SREFP 3 C00091 BC00091  +REFP EC00091
CALL JOB:SEARCH-R1-S13D
SET P023 P006
SFTON3D P023
SMOVL C00092 BC00092 V=166.7  +MOVJ EC00092
SMOVL C00093 BC00093 V=500.0  +MOVJ EC00093
SMOVL C00094 BC00094 V=166.7  +MOVJ EC00094
SREFP 3 C00095 BC00095  +REFP EC00095
CALL JOB:SEARCH-R1-S13D
SET P023 P006
SFTON3D P023
SMOVL C00096 BC00096 V=166.7  +MOVJ EC00096
SMOVL C00097 BC00097 V=166.7  +MOVJ EC00097
SREFP 3 C00098 BC00098  +REFP EC00098
CALL JOB:SEARCH-R1-S13D
SET P023 P006
SFTON3D P023
SMOVL C00099 BC00099 V=166.7  +MOVJ EC00099
MOVL C00100 BC00100 V=1000.0  +MOVJ EC00100 VJ=100.00
MOVJ C00101 BC00101 VJ=80.00  +MOVJ EC00101 VJ=80.00
MOVJ C00102 BC00102 VJ=80.00  +MOVJ EC00102 VJ=80.00
SFTOF3D
MOVJ C00103 BC00103 VJ=80.00  +MOVJ EC00103 VJ=80.00
SMOVL C00104 BC00104 V=166.7  +MOVJ EC00104
SREFP 3 C00105 BC00105  +REFP EC00105
CALL JOB:SEARCH-R1-S13D
SET P061 P006
SFTON3D P061
SMOVL C00106 BC00106 V=166.7  +MOVJ EC00106
SREFP 3 C00107 BC00107  +REFP EC00107
CALL JOB:SEARCH-R1-S13D
SET P061 P006
SFTON3D P061
SMOVL C00108 BC00108 V=166.7  +MOVJ EC00108
SFTOF3D
SMOVL C00109 BC00109 V=500.0  +MOVJ EC00109
SMOVL C00110 BC00110 V=166.7  +MOVJ EC00110
SREFP 3 C00111 BC00111  +REFP EC00111
CALL JOB:SEARCH-R1-S13D
SET P062 P006
SFTON3D P062
SMOVL C00112 BC00112 V=166.7  +MOVJ EC00112
SREFP 3 C00113 BC00113  +REFP EC00113
CALL JOB:SEARCH-R1-S13D
SET P062 P006
SFTON3D P062
SMOVL C00114 BC00114 V=166.7  +MOVJ EC00114
SFTOF3D
SMOVL C00115 BC00115 V=500.0  +MOVJ EC00115
SMOVL C00116 BC00116 V=166.7  +MOVJ EC00116
SREFP 3 C00117 BC00117  +REFP EC00117
CALL JOB:SEARCH-R1-S13D
SET P063 P006
SFTON3D P063
SMOVL C00118 BC00118 V=166.7  +MOVJ EC00118
SREFP 3 C00119 BC00119  +REFP EC00119
CALL JOB:SEARCH-R1-S13D
SET P063 P006
SFTON3D P063
SMOVL C00120 BC00120 V=166.7  +MOVJ EC00120
SFTOF3D
SMOVL C00121 BC00121 V=500.0  +MOVJ EC00121
MOVJ C00122 BC00122 VJ=80.00  +MOVJ EC00122 VJ=80.00
MOVJ C00123 BC00123 VJ=80.00  +MOVJ EC00123 VJ=80.00
'EndPath S3464
MOVJ C00124 BC00124 VJ=100.00  +MOVJ EC00124 VJ=100.00
'Path S3465
SFTOF3D
MOVJ C00125 BC00125 VJ=100.00  +MOVJ EC00125 VJ=100.00
MOVL C00126 BC00126 V=666.7  +MOVJ EC00126 VJ=100.00
SMOVL C00127 BC00127 V=166.7  +MOVJ EC00127
SREFP 3 C00128 BC00128  +REFP EC00128
CALL JOB:SEARCH-R1-S13D
SET P024 P006
SFTON3D P024
SMOVL C00129 BC00129 V=166.7  +MOVJ EC00129
SREFP 3 C00130 BC00130  +REFP EC00130
CALL JOB:SEARCH-R1-S13D
SET P024 P006
SFTON3D P024
SMOVL C00131 BC00131 V=166.7  +MOVJ EC00131
SMOVL C00132 BC00132 V=166.7  +MOVJ EC00132
SREFP 3 C00133 BC00133  +REFP EC00133
CALL JOB:SEARCH-R1-S13D
SET P024 P006
SFTON3D P024
SMOVL C00134 BC00134 V=166.7  +MOVJ EC00134
MOVL C00135 BC00135 V=1000.0  +MOVJ EC00135 VJ=100.00
'EndPath S3465
'Path S3476
SFTOF3D
MOVJ C00136 BC00136 VJ=100.00  +MOVJ EC00136 VJ=100.00
MOVL C00137 BC00137 V=666.7  +MOVJ EC00137 VJ=100.00
SMOVL C00138 BC00138 V=166.7  +MOVJ EC00138
SREFP 3 C00139 BC00139  +REFP EC00139
CALL JOB:SEARCH-R1-S13D
SET P035 P006
SFTON3D P035
SMOVL C00140 BC00140 V=166.7  +MOVJ EC00140
SREFP 3 C00141 BC00141  +REFP EC00141
CALL JOB:SEARCH-R1-S13D
SET P035 P006
SFTON3D P035
SMOVL C00142 BC00142 V=166.7  +MOVJ EC00142
SMOVL C00143 BC00143 V=333.3  +MOVJ EC00143
SMOVL C00144 BC00144 V=166.7  +MOVJ EC00144
SREFP 3 C00145 BC00145  +REFP EC00145
CALL JOB:SEARCH-R1-S13D
SET P035 P006
SFTON3D P035
SMOVL C00146 BC00146 V=166.7  +MOVJ EC00146
MOVL C00147 BC00147 V=1000.0  +MOVJ EC00147 VJ=100.00
'EndPath S3476
'Path S3470
SFTOF3D
MOVJ C00148 BC00148 VJ=100.00  +MOVJ EC00148 VJ=100.00
MOVL C00149 BC00149 V=666.7  +MOVJ EC00149 VJ=100.00
SMOVL C00150 BC00150 V=166.7  +MOVJ EC00150
SREFP 3 C00151 BC00151  +REFP EC00151
CALL JOB:SEARCH-R1-S13D
SET P029 P006
SFTON3D P029
SMOVL C00152 BC00152 V=166.7  +MOVJ EC00152
SREFP 3 C00153 BC00153  +REFP EC00153
CALL JOB:SEARCH-R1-S13D
SET P029 P006
SFTON3D P029
SMOVL C00154 BC00154 V=166.7  +MOVJ EC00154
SMOVL C00155 BC00155 V=250.0  +MOVJ EC00155
SMOVL C00156 BC00156 V=166.7  +MOVJ EC00156
SREFP 3 C00157 BC00157  +REFP EC00157
CALL JOB:SEARCH-R1-S13D
SET P029 P006
SFTON3D P029
SMOVL C00158 BC00158 V=166.7  +MOVJ EC00158
MOVL C00159 BC00159 V=1000.0  +MOVJ EC00159 VJ=100.00
'EndPath S3470
'Path S4850
SFTOF3D
MOVL C00160 BC00160 V=666.7  +MOVJ EC00160 VJ=100.00
SMOVL C00161 BC00161 V=166.7  +MOVJ EC00161
SREFP 3 C00162 BC00162  +REFP EC00162
CALL JOB:SEARCH-R1-S13D
SET P071 P006
SFTON3D P071
SMOVL C00163 BC00163 V=166.7  +MOVJ EC00163
SREFP 3 C00164 BC00164  +REFP EC00164
CALL JOB:SEARCH-R1-S13D
SET P071 P006
SFTON3D P071
SMOVL C00165 BC00165 V=166.7  +MOVJ EC00165
SMOVL C00166 BC00166 V=166.7  +MOVJ EC00166
SREFP 3 C00167 BC00167  +REFP EC00167
CALL JOB:SEARCH-R1-S13D
SET P071 P006
SFTON3D P071
SMOVL C00168 BC00168 V=166.7  +MOVJ EC00168
MOVL C00169 BC00169 V=1000.0  +MOVJ EC00169 VJ=100.00
'EndPath S4850
'Path S4851
SFTOF3D
MOVJ C00170 BC00170 VJ=100.00  +MOVJ EC00170 VJ=100.00
MOVL C00171 BC00171 V=666.7  +MOVJ EC00171 VJ=100.00
SMOVL C00172 BC00172 V=166.7  +MOVJ EC00172
SREFP 3 C00173 BC00173  +REFP EC00173
CALL JOB:SEARCH-R1-S13D
SET P072 P006
SFTON3D P072
SMOVL C00174 BC00174 V=166.7  +MOVJ EC00174
SREFP 3 C00175 BC00175  +REFP EC00175
CALL JOB:SEARCH-R1-S13D
SET P072 P006
SFTON3D P072
SMOVL C00176 BC00176 V=166.7  +MOVJ EC00176
MOVL C00177 BC00177 V=1000.0  +MOVJ EC00177 VJ=100.00
'EndPath S4851
MOVJ C00178 BC00178 VJ=100.00  +MOVJ EC00178 VJ=100.00
MOVJ C00179 BC00179 VJ=100.00  +MOVJ EC00179 VJ=100.00
'Path S4852
SFTOF3D
MOVJ C00180 BC00180 VJ=100.00  +MOVJ EC00180 VJ=100.00
MOVL C00181 BC00181 V=666.7  +MOVJ EC00181 VJ=100.00
SMOVL C00182 BC00182 V=166.7  +MOVJ EC00182
SREFP 3 C00183 BC00183  +REFP EC00183
CALL JOB:SEARCH-R1-S13D
SET P073 P006
SFTON3D P073
SMOVL C00184 BC00184 V=166.7  +MOVJ EC00184
SMOVL C00185 BC00185 V=166.7  +MOVJ EC00185
SREFP 3 C00186 BC00186  +REFP EC00186
CALL JOB:SEARCH-R1-S13D
SET P073 P006
SFTON3D P073
SMOVL C00187 BC00187 V=166.7  +MOVJ EC00187
SMOVL C00188 BC00188 V=166.7  +MOVJ EC00188
SREFP 3 C00189 BC00189  +REFP EC00189
CALL JOB:SEARCH-R1-S13D
SET P073 P006
SFTON3D P073
SMOVL C00190 BC00190 V=166.7  +MOVJ EC00190
MOVL C00191 BC00191 V=1000.0  +MOVJ EC00191 VJ=100.00
'EndPath S4852
MOVJ C00192 BC00192 VJ=100.00  +MOVJ EC00192 VJ=100.00
'Path S4853
SFTOF3D
MOVJ C00193 BC00193 VJ=100.00  +MOVJ EC00193 VJ=100.00
MOVL C00194 BC00194 V=666.7  +MOVJ EC00194 VJ=100.00
SMOVL C00195 BC00195 V=166.7  +MOVJ EC00195
SREFP 3 C00196 BC00196  +REFP EC00196
CALL JOB:SEARCH-R1-S13D
SET P074 P006
SFTON3D P074
SMOVL C00197 BC00197 V=166.7  +MOVJ EC00197
SREFP 3 C00198 BC00198  +REFP EC00198
CALL JOB:SEARCH-R1-S13D
SET P074 P006
SFTON3D P074
SMOVL C00199 BC00199 V=166.7  +MOVJ EC00199
MOVL C00200 BC00200 V=1000.0  +MOVJ EC00200 VJ=100.00
'EndPath S4853
'Path S3467
SFTOF3D
MOVJ C00201 BC00201 VJ=100.00  +MOVJ EC00201 VJ=100.00
MOVJ C00202 BC00202 VJ=50.00  +MOVJ EC00202 VJ=50.00
MOVJ C00203 BC00203 VJ=100.00  +MOVJ EC00203 VJ=100.00
MOVJ C00204 BC00204 VJ=100.00  +MOVJ EC00204 VJ=100.00
MOVL C00205 BC00205 V=666.7  +MOVJ EC00205 VJ=100.00
SMOVL C00206 BC00206 V=166.7  +MOVJ EC00206
SREFP 3 C00207 BC00207  +REFP EC00207
CALL JOB:SEARCH-R1-S13D
SET P026 P006
SFTON3D P026
SMOVL C00208 BC00208 V=166.7  +MOVJ EC00208
SREFP 3 C00209 BC00209  +REFP EC00209
CALL JOB:SEARCH-R1-S13D
SET P026 P006
SFTON3D P026
SMOVL C00210 BC00210 V=166.7  +MOVJ EC00210
SMOVL C00211 BC00211 V=800.0  +MOVJ EC00211
SMOVL C00212 BC00212 V=166.7  +MOVJ EC00212
SREFP 3 C00213 BC00213  +REFP EC00213
CALL JOB:SEARCH-R1-S13D
SET P026 P006
SFTON3D P026
SMOVL C00214 BC00214 V=166.7  +MOVJ EC00214
MOVL C00215 BC00215 V=1000.0  +MOVJ EC00215 VJ=100.00
'EndPath S3467
MOVJ C00216 BC00216 VJ=100.00  +MOVJ EC00216 VJ=100.00
'Path S3466
SFTOF3D
MOVJ C00217 BC00217 VJ=100.00  +MOVJ EC00217 VJ=100.00
MOVL C00218 BC00218 V=666.7  +MOVJ EC00218 VJ=100.00
SMOVL C00219 BC00219 V=166.7  +MOVJ EC00219
SREFP 3 C00220 BC00220  +REFP EC00220
CALL JOB:SEARCH-R1-S13D
SET P025 P006
SFTON3D P025
SMOVL C00221 BC00221 V=166.7  +MOVJ EC00221
SMOVL C00222 BC00222 V=166.7  +MOVJ EC00222
SREFP 3 C00223 BC00223  +REFP EC00223
CALL JOB:SEARCH-R1-S13D
SET P025 P006
SFTON3D P025
SMOVL C00224 BC00224 V=166.7  +MOVJ EC00224
SMOVL C00225 BC00225 V=200.0  +MOVJ EC00225
SMOVL C00226 BC00226 V=166.7  +MOVJ EC00226
SREFP 3 C00227 BC00227  +REFP EC00227
CALL JOB:SEARCH-R1-S13D
SET P025 P006
SFTON3D P025
SMOVL C00228 BC00228 V=166.7  +MOVJ EC00228
MOVL C00229 BC00229 V=1000.0  +MOVJ EC00229 VJ=100.00
'EndPath S3466
MOVJ C00230 BC00230 VJ=100.00  +MOVJ EC00230 VJ=100.00
'Path S3469
SFTOF3D
MOVJ C00231 BC00231 VJ=100.00  +MOVJ EC00231 VJ=100.00
MOVL C00232 BC00232 V=666.7  +MOVJ EC00232 VJ=100.00
SMOVL C00233 BC00233 V=166.7  +MOVJ EC00233
SREFP 3 C00234 BC00234  +REFP EC00234
CALL JOB:SEARCH-R1-S13D
SET P028 P006
SFTON3D P028
SMOVL C00235 BC00235 V=166.7  +MOVJ EC00235
SREFP 3 C00236 BC00236  +REFP EC00236
CALL JOB:SEARCH-R1-S13D
SET P028 P006
SFTON3D P028
SMOVL C00237 BC00237 V=166.7  +MOVJ EC00237
SMOVL C00238 BC00238 V=333.3  +MOVJ EC00238
SMOVL C00239 BC00239 V=166.7  +MOVJ EC00239
SREFP 3 C00240 BC00240  +REFP EC00240
CALL JOB:SEARCH-R1-S13D
SET P028 P006
SFTON3D P028
SMOVL C00241 BC00241 V=166.7  +MOVJ EC00241
MOVL C00242 BC00242 V=1000.0  +MOVJ EC00242 VJ=100.00
'EndPath S3469
MOVJ C00243 BC00243 VJ=100.00  +MOVJ EC00243 VJ=100.00
'Path S3474
SFTOF3D
MOVJ C00244 BC00244 VJ=100.00  +MOVJ EC00244 VJ=100.00
MOVL C00245 BC00245 V=666.7  +MOVJ EC00245 VJ=100.00
SMOVL C00246 BC00246 V=166.7  +MOVJ EC00246
SREFP 3 C00247 BC00247  +REFP EC00247
CALL JOB:SEARCH-R1-S13D
SET P033 P006
SFTON3D P033
SMOVL C00248 BC00248 V=166.7  +MOVJ EC00248
SREFP 3 C00249 BC00249  +REFP EC00249
CALL JOB:SEARCH-R1-S13D
SET P033 P006
SFTON3D P033
SMOVL C00250 BC00250 V=166.7  +MOVJ EC00250
SMOVL C00251 BC00251 V=250.0  +MOVJ EC00251
SMOVL C00252 BC00252 V=166.7  +MOVJ EC00252
SREFP 3 C00253 BC00253  +REFP EC00253
CALL JOB:SEARCH-R1-S13D
SET P033 P006
SFTON3D P033
SMOVL C00254 BC00254 V=166.7  +MOVJ EC00254
MOVL C00255 BC00255 V=1000.0  +MOVJ EC00255 VJ=100.00
'EndPath S3474
'Path S3468
SFTOF3D
MOVJ C00256 BC00256 VJ=100.00  +MOVJ EC00256 VJ=100.00
MOVL C00257 BC00257 V=666.7  +MOVJ EC00257 VJ=100.00
SMOVL C00258 BC00258 V=166.7  +MOVJ EC00258
SREFP 3 C00259 BC00259  +REFP EC00259
CALL JOB:SEARCH-R1-S13D
SET P027 P006
SFTON3D P027
SMOVL C00260 BC00260 V=166.7  +MOVJ EC00260
SMOVL C00261 BC00261 V=166.7  +MOVJ EC00261
SREFP 3 C00262 BC00262  +REFP EC00262
CALL JOB:SEARCH-R1-S13D
SET P027 P006
SFTON3D P027
SMOVL C00263 BC00263 V=166.7  +MOVJ EC00263
SMOVL C00264 BC00264 V=166.7  +MOVJ EC00264
SREFP 3 C00265 BC00265  +REFP EC00265
CALL JOB:SEARCH-R1-S13D
SET P027 P006
SFTON3D P027
SMOVL C00266 BC00266 V=166.7  +MOVJ EC00266
MOVL C00267 BC00267 V=1000.0  +MOVJ EC00267 VJ=100.00
'EndPath S3468
'Path S3471
SFTOF3D
MOVJ C00268 BC00268 VJ=100.00  +MOVJ EC00268 VJ=100.00
MOVL C00269 BC00269 V=666.7  +MOVJ EC00269 VJ=100.00
SMOVL C00270 BC00270 V=166.7  +MOVJ EC00270
SREFP 3 C00271 BC00271  +REFP EC00271
CALL JOB:SEARCH-R1-S13D
SET P030 P006
SFTON3D P030
SMOVL C00272 BC00272 V=166.7  +MOVJ EC00272
SREFP 3 C00273 BC00273  +REFP EC00273
CALL JOB:SEARCH-R1-S13D
SET P030 P006
SFTON3D P030
SMOVL C00274 BC00274 V=166.7  +MOVJ EC00274
MOVL C00275 BC00275 V=1000.0  +MOVJ EC00275 VJ=100.00
'EndPath S3471
'Path S3472
SFTOF3D
MOVJ C00276 BC00276 VJ=100.00  +MOVJ EC00276 VJ=100.00
MOVL C00277 BC00277 V=666.7  +MOVJ EC00277 VJ=100.00
SMOVL C00278 BC00278 V=166.7  +MOVJ EC00278
SREFP 3 C00279 BC00279  +REFP EC00279
CALL JOB:SEARCH-R1-S13D
SET P031 P006
SFTON3D P031
SMOVL C00280 BC00280 V=166.7  +MOVJ EC00280
SREFP 3 C00281 BC00281  +REFP EC00281
CALL JOB:SEARCH-R1-S13D
SET P031 P006
SFTON3D P031
SMOVL C00282 BC00282 V=166.7  +MOVJ EC00282
MOVL C00283 BC00283 V=1000.0  +MOVJ EC00283 VJ=100.00
'EndPath S3472
MOVJ C00284 BC00284 VJ=100.00  +MOVJ EC00284 VJ=100.00
'Path S3472
SFTOF3D
MOVJ C00285 BC00285 VJ=100.00  +MOVJ EC00285 VJ=100.00
MOVL C00286 BC00286 V=666.7  +MOVJ EC00286 VJ=100.00
SMOVL C00287 BC00287 V=166.7  +MOVJ EC00287
SREFP 3 C00288 BC00288  +REFP EC00288
CALL JOB:SEARCH-R1-S13D
SET P032 P006
SFTON3D P032
SMOVL C00289 BC00289 V=166.7  +MOVJ EC00289
SREFP 3 C00290 BC00290  +REFP EC00290
CALL JOB:SEARCH-R1-S13D
SET P032 P006
SFTON3D P032
SMOVL C00291 BC00291 V=166.7  +MOVJ EC00291
SMOVL C00292 BC00292 V=133.3  +MOVJ EC00292
SREFP 3 C00293 BC00293  +REFP EC00293
CALL JOB:SEARCH-R1-S13D
SET P032 P006
SFTON3D P032
SMOVL C00294 BC00294 V=166.7  +MOVJ EC00294
MOVL C00295 BC00295 V=1000.0  +MOVJ EC00295 VJ=100.00
'EndPath S3472
MOVJ C00296 BC00296 VJ=100.00  +MOVJ EC00296 VJ=100.00
'Path S3477
SFTOF3D
MOVJ C00297 BC00297 VJ=100.00  +MOVJ EC00297 VJ=100.00
SMOVL C00298 BC00298 V=166.7  +MOVJ EC00298
SREFP 3 C00299 BC00299  +REFP EC00299
CALL JOB:SEARCH-R1-S13D
SET P069 P006
SFTON3D P069
SMOVL C00300 BC00300 V=250.0  +MOVJ EC00300
SMOVL C00301 BC00301 V=250.0  +MOVJ EC00301
SMOVL C00302 BC00302 V=166.7  +MOVJ EC00302
SREFP 3 C00303 BC00303  +REFP EC00303
CALL JOB:SEARCH-R1-S13D
SET P069 P006
SFTON3D P069
SMOVL C00304 BC00304 V=166.7  +MOVJ EC00304
SFTOF3D
SMOVL C00305 BC00305 V=666.7  +MOVJ EC00305
MOVL C00306 BC00306 V=666.7  +MOVJ EC00306 VJ=100.00
SMOVL C00307 BC00307 V=166.7  +MOVJ EC00307
SREFP 3 C00308 BC00308  +REFP EC00308
CALL JOB:SEARCH-R1-S13D
SET P052 P006
SFTON3D P052
SMOVL C00309 BC00309 V=166.7  +MOVJ EC00309
SREFP 3 C00310 BC00310  +REFP EC00310
CALL JOB:SEARCH-R1-S13D
SET P052 P006
SFTON3D P052
SMOVL C00311 BC00311 V=166.7  +MOVJ EC00311
MOVL C00312 BC00312 V=1000.0  +MOVJ EC00312 VJ=100.00
'EndPath S3477
MOVJ C00313 BC00313 VJ=100.00  +MOVJ EC00313 VJ=100.00
'poprawiÄ searcha- nie mialem
'wyciecia
'Path S3478
SFTOF3D
MOVJ C00314 BC00314 VJ=100.00  +MOVJ EC00314 VJ=100.00
MOVL C00315 BC00315 V=666.7  +MOVJ EC00315 VJ=100.00
SMOVL C00316 BC00316 V=166.7  +MOVJ EC00316
SREFP 3 C00317 BC00317  +REFP EC00317
CALL JOB:SEARCH-R1-S13D
SET P053 P006
SFTON3D P053
SMOVL C00318 BC00318 V=166.7  +MOVJ EC00318
SREFP 3 C00319 BC00319  +REFP EC00319
CALL JOB:SEARCH-R1-S13D
SET P053 P006
SFTON3D P053
SMOVL C00320 BC00320 V=166.7  +MOVJ EC00320
MOVL C00321 BC00321 V=1000.0  +MOVJ EC00321 VJ=100.00
'EndPath S3478
'
MOVJ C00322 BC00322 VJ=100.00  +MOVJ EC00322 VJ=100.00
'Path W3476
SFTOF3D
SFTON3D P033
MOVJ C00323 BC00323 VJ=100.00  +MOVJ EC00323 VJ=100.00
SMOVL C00324 BC00324 V=800.0  +MOVJ EC00324
SMOVL C00325 BC00325 V=166.7 PL=0  +MOVJ EC00325
MACRO1 MJ#(0) ARGF14
ARCON
SMOVL C00326 BC00326 V=10.0  +MOVJ EC00326
ARCOF
SMOVL C00327 BC00327 V=800.0  +MOVJ EC00327
SMOVL C00328 BC00328 V=1000.0  +MOVJ EC00328
SFTOF3D
'EndPath W3476
'Path W3477
SFTOF3D
SFTON3D P033
MOVJ C00329 BC00329 VJ=100.00  +MOVJ EC00329 VJ=100.00
SMOVL C00330 BC00330 V=800.0  +MOVJ EC00330
SMOVL C00331 BC00331 V=166.7 PL=0  +MOVJ EC00331
SMOVL C00332 BC00332 V=10.0  +MOVJ EC00332
SMOVL C00333 BC00333 V=10.0  +MOVJ EC00333
SMOVL C00334 BC00334 V=10.0  +MOVJ EC00334
ARCOF
SMOVL C00335 BC00335 V=800.0  +MOVJ EC00335
SMOVL C00336 BC00336 V=1000.0  +MOVJ EC00336
SFTOF3D
'EndPath W3477
MOVJ C00337 BC00337 VJ=100.00  +MOVJ EC00337 VJ=100.00
'Path W3478
SFTOF3D
SFTON3D P033
MOVJ C00338 BC00338 VJ=100.00  +MOVJ EC00338 VJ=100.00
SMOVL C00339 BC00339 V=800.0  +MOVJ EC00339
SMOVL C00340 BC00340 V=166.7 PL=0  +MOVJ EC00340
ARCON
SMOVL C00341 BC00341 V=10.0  +MOVJ EC00341
SMOVL C00342 BC00342 V=10.0  +MOVJ EC00342
SMOVL C00343 BC00343 V=10.0  +MOVJ EC00343
ARCOF
SMOVL C00344 BC00344 V=800.0  +MOVJ EC00344
SMOVL C00345 BC00345 V=1000.0  +MOVJ EC00345
SFTOF3D
'EndPath W3478
MOVJ C00346 BC00346 VJ=100.00  +MOVJ EC00346 VJ=100.00
MOVJ C00347 BC00347 VJ=100.00  +MOVJ EC00347 VJ=100.00
'9
'Path W3479
SFTOF3D
SFTON3D P026
MOVJ C00348 BC00348 VJ=100.00  +MOVJ EC00348 VJ=100.00
SMOVL C00349 BC00349 V=800.0  +MOVJ EC00349
SMOVL C00350 BC00350 V=166.7 PL=0  +MOVJ EC00350
ARCON
SMOVL C00351 BC00351 V=9.2  +MOVJ EC00351
SMOVL C00352 BC00352 V=9.2  +MOVJ EC00352
SMOVL C00353 BC00353 V=9.2  +MOVJ EC00353
ARCOF
SMOVL C00354 BC00354 V=800.0  +MOVJ EC00354
SMOVL C00355 BC00355 V=1000.0  +MOVJ EC00355
SFTOF3D
'EndPath W3479
'Path W3480
SFTOF3D
SFTON3D P026
MOVJ C00356 BC00356 VJ=100.00  +MOVJ EC00356 VJ=100.00
SMOVL C00357 BC00357 V=800.0  +MOVJ EC00357
SMOVL C00358 BC00358 V=150.0 PL=0  +MOVJ EC00358
ARCON
SMOVL C00359 BC00359 V=10.0  +MOVJ EC00359
SMOVL C00360 BC00360 V=10.0  +MOVJ EC00360
SMOVL C00361 BC00361 V=10.0  +MOVJ EC00361
ARCOF
SMOVL C00362 BC00362 V=800.0  +MOVJ EC00362
SMOVL C00363 BC00363 V=1000.0  +MOVJ EC00363
SFTOF3D
'EndPath W3480
'Path W3481
SFTOF3D
SFTON3D P026
MOVJ C00364 BC00364 VJ=100.00  +MOVJ EC00364 VJ=100.00
SMOVL C00365 BC00365 V=800.0  +MOVJ EC00365
SMOVL C00366 BC00366 V=150.0 PL=0  +MOVJ EC00366
SMOVL C00367 BC00367 V=10.0  +MOVJ EC00367
ARCOF
SMOVL C00368 BC00368 V=800.0  +MOVJ EC00368
SMOVL C00369 BC00369 V=1000.0  +MOVJ EC00369
SFTOF3D
'EndPath W3481
MOVJ C00370 BC00370 VJ=100.00  +MOVJ EC00370 VJ=100.00
'uwaga na podajnik
'Path W3481
SFTOF3D
SFTON3D P026
MOVJ C00371 BC00371 VJ=50.00  +MOVJ EC00371 VJ=15.00
SMOVL C00372 BC00372 V=800.0  +MOVJ EC00372
SMOVL C00373 BC00373 V=150.0 PL=0  +MOVJ EC00373
ARCON
SMOVL C00374 BC00374 V=10.0  +MOVJ EC00374
SMOVL C00375 BC00375 V=10.0  +MOVJ EC00375
ARCOF
SMOVL C00376 BC00376 V=800.0  +MOVJ EC00376
SMOVL C00377 BC00377 V=1000.0  +MOVJ EC00377
SFTOF3D
'EndPath W3481
'brak dostepu offset drutu 1cm
'Path W3482
SFTOF3D
SFTON3D P026
MOVJ C00378 BC00378 VJ=100.00  +MOVJ EC00378 VJ=100.00
SMOVL C00379 BC00379 V=800.0  +MOVJ EC00379
SMOVL C00380 BC00380 V=150.0 PL=0  +MOVJ EC00380
ARCON
SMOVL C00381 BC00381 V=10.0  +MOVJ EC00381
ARCOF
SMOVL C00382 BC00382 V=800.0  +MOVJ EC00382
SMOVL C00383 BC00383 V=1000.0  +MOVJ EC00383
SFTOF3D
'EndPath W3482
MOVJ C00384 BC00384 VJ=100.00  +MOVJ EC00384 VJ=100.00
MOVJ C00385 BC00385 VJ=100.00  +MOVJ EC00385 VJ=100.00
'10
'11
'Path W3484
SFTOF3D
SFTON3D P025
MOVJ C00386 BC00386 VJ=100.00  +MOVJ EC00386 VJ=100.00
SMOVL C00387 BC00387 V=800.0  +MOVJ EC00387
SMOVL C00388 BC00388 V=150.0 PL=0  +MOVJ EC00388
ARCON
SMOVL C00389 BC00389 V=10.0  +MOVJ EC00389
SMOVL C00390 BC00390 V=10.0  +MOVJ EC00390
ARCOF
SMOVL C00391 BC00391 V=800.0  +MOVJ EC00391
SMOVL C00392 BC00392 V=1000.0  +MOVJ EC00392
SFTOF3D
'EndPath W3484
MOVJ C00393 BC00393 VJ=100.00  +MOVJ EC00393 VJ=100.00
'brak dostepu offset drutu 1cm
'Path W3483
SFTOF3D
SFTON3D P025
MOVJ C00394 BC00394 VJ=100.00  +MOVJ EC00394 VJ=100.00
SMOVL C00395 BC00395 V=800.0  +MOVJ EC00395
SMOVL C00396 BC00396 V=166.7 PL=0  +MOVJ EC00396
ARCON
SMOVL C00397 BC00397 V=10.0  +MOVJ EC00397
ARCOF
SMOVL C00398 BC00398 V=800.0  +MOVJ EC00398
SMOVL C00399 BC00399 V=1000.0  +MOVJ EC00399
SFTOF3D
'EndPath W3483
MOVJ C00400 BC00400 VJ=100.00  +MOVJ EC00400 VJ=100.00
MOVJ C00401 BC00401 VJ=100.00  +MOVJ EC00401 VJ=100.00
MOVJ C00402 BC00402 VJ=100.00  +MOVJ EC00402 VJ=100.00
'Path W4854
SFTOF3D
SFTON3D P073
MOVJ C00403 BC00403 VJ=100.00  +MOVJ EC00403 VJ=100.00
SMOVL C00404 BC00404 V=800.0  +MOVJ EC00404
SMOVL C00405 BC00405 V=150.0 PL=0  +MOVJ EC00405
MACRO1 MJ#(0) ARGF9
ARCON
SMOVL C00406 BC00406 V=9.2  +MOVJ EC00406
SFTON3D P074
SMOVL C00407 BC00407 V=9.2  +MOVJ EC00407
SMOVL C00408 BC00408 V=9.2  +MOVJ EC00408
ARCOF
SMOVL C00409 BC00409 V=800.0  +MOVJ EC00409
SMOVL C00410 BC00410 V=1000.0  +MOVJ EC00410
SFTOF3D
'EndPath W4854
'12
MOVJ C00411 BC00411 VJ=100.00  +MOVJ EC00411 VJ=100.00
MOVJ C00412 BC00412 VJ=100.00  +MOVJ EC00412 VJ=100.00
MOVJ C00413 BC00413 VJ=100.00  +MOVJ EC00413 VJ=100.00
'Path W3485
SFTOF3D
SFTON3D P034
MOVJ C00414 BC00414 VJ=100.00  +MOVJ EC00414 VJ=100.00
SMOVL C00415 BC00415 V=800.0  +MOVJ EC00415
SMOVL C00416 BC00416 V=150.0 PL=0  +MOVJ EC00416
MACRO1 MJ#(0) ARGF14
ARCON
SMOVL C00417 BC00417 V=10.0  +MOVJ EC00417
SMOVL C00418 BC00418 V=10.0  +MOVJ EC00418
SMOVL C00419 BC00419 V=10.0  +MOVJ EC00419
ARCOF
SMOVL C00420 BC00420 V=800.0  +MOVJ EC00420
SMOVL C00421 BC00421 V=1000.0  +MOVJ EC00421
SFTOF3D
MOVJ C00422 BC00422 VJ=80.00  +MOVJ EC00422 VJ=80.00
MOVJ C00423 BC00423 VJ=80.00  +MOVJ EC00423 VJ=80.00
MOVJ C00424 BC00424 VJ=80.00  +MOVJ EC00424 VJ=80.00
MACRO1 MJ#(0) ARGF6
SFTON3D P063
SMOVL C00425 BC00425 V=166.7  +MOVJ EC00425
ARCON
SMOVL C00426 BC00426 V=11.7  +MOVJ EC00426
SMOVL C00427 BC00427 V=11.7  +MOVJ EC00427
SFTON3D P062
SMOVL C00428 BC00428 V=11.0  +MOVJ EC00428
SMOVL C00429 BC00429 V=11.0  +MOVJ EC00429
SFTON3D P061
SMOVL C00430 BC00430 V=11.0  +MOVJ EC00430
SMOVL C00431 BC00431 V=11.0  +MOVJ EC00431
ARCOF
SMOVL C00432 BC00432 V=800.0  +MOVJ EC00432
SFTOF3D
MOVJ C00433 BC00433 VJ=80.00  +MOVJ EC00433 VJ=80.00
MOVJ C00434 BC00434 VJ=80.00  +MOVJ EC00434 VJ=80.00
MOVJ C00435 BC00435 VJ=80.00  +MOVJ EC00435 VJ=80.00
'EndPath W3485
'Path W3486
SFTOF3D
SFTON3D P050
MOVJ C00436 BC00436 VJ=100.00  +MOVJ EC00436 VJ=100.00
SMOVL C00437 BC00437 V=800.0  +MOVJ EC00437
SMOVL C00438 BC00438 V=150.0 PL=0  +MOVJ EC00438
MACRO1 MJ#(0) ARGF14
ARCON
SMOVL C00439 BC00439 V=10.0  +MOVJ EC00439
SMOVL C00440 BC00440 V=10.0  +MOVJ EC00440
SMOVL C00441 BC00441 V=10.0  +MOVJ EC00441
ARCOF
SMOVL C00442 BC00442 V=800.0  +MOVJ EC00442
SMOVL C00443 BC00443 V=1000.0  +MOVJ EC00443
SFTOF3D
'EndPath W3486
MOVJ C00444 BC00444 VJ=100.00  +MOVJ EC00444 VJ=100.00
'Path W3485
SFTOF3D
SFTON3D P034
MOVJ C00445 BC00445 VJ=100.00  +MOVJ EC00445 VJ=100.00
SMOVL C00446 BC00446 V=800.0  +MOVJ EC00446
SMOVL C00447 BC00447 V=166.7 PL=0  +MOVJ EC00447
ARCON
SMOVL C00448 BC00448 V=9.2  +MOVJ EC00448
SMOVL C00449 BC00449 V=9.2  +MOVJ EC00449
SMOVL C00450 BC00450 V=9.2  +MOVJ EC00450
ARCOF
SMOVL C00451 BC00451 V=800.0  +MOVJ EC00451
SMOVL C00452 BC00452 V=1000.0  +MOVJ EC00452
SFTOF3D
'EndPath W3485
'Path W3487
SFTOF3D
SFTON3D P054
MOVJ C00453 BC00453 VJ=100.00  +MOVJ EC00453 VJ=100.00
SMOVL C00454 BC00454 V=800.0  +MOVJ EC00454
SMOVL C00455 BC00455 V=150.0 PL=0  +MOVJ EC00455
ARCON
SMOVL C00456 BC00456 V=9.2  +MOVJ EC00456
SMOVL C00457 BC00457 V=9.2  +MOVJ EC00457
SMOVL C00458 BC00458 V=9.2  +MOVJ EC00458
ARCOF
SMOVL C00459 BC00459 V=800.0  +MOVJ EC00459
SMOVL C00460 BC00460 V=1000.0  +MOVJ EC00460
SFTOF3D
'EndPath W3487
MOVJ C00461 BC00461 VJ=100.00  +MOVJ EC00461 VJ=100.00
'Path W3487
SFTOF3D
SFTON3D P028
MOVJ C00462 BC00462 VJ=100.00  +MOVJ EC00462 VJ=100.00
SMOVL C00463 BC00463 V=800.0  +MOVJ EC00463
SMOVL C00464 BC00464 V=150.0 PL=0  +MOVJ EC00464
ARCON
SMOVL C00465 BC00465 V=9.2  +MOVJ EC00465
SMOVL C00466 BC00466 V=9.2  +MOVJ EC00466
SMOVL C00467 BC00467 V=9.2  +MOVJ EC00467
ARCOF
SMOVL C00468 BC00468 V=800.0  +MOVJ EC00468
SMOVL C00469 BC00469 V=1000.0  +MOVJ EC00469
SFTOF3D
'EndPath W3487
MOVJ C00470 BC00470 VJ=100.00  +MOVJ EC00470 VJ=100.00
MOVJ C00471 BC00471 VJ=100.00  +MOVJ EC00471 VJ=100.00
'brak dostepu offset 5mm
'Path W3488
SFTOF3D
SFTON3D P028
MOVJ C00472 BC00472 VJ=100.00  +MOVJ EC00472 VJ=100.00
SMOVL C00473 BC00473 V=800.0  +MOVJ EC00473
SMOVL C00474 BC00474 V=150.0 PL=0  +MOVJ EC00474
ARCON
SMOVL C00475 BC00475 V=11.7  +MOVJ EC00475
ARCOF
SMOVL C00476 BC00476 V=800.0  +MOVJ EC00476
SMOVL C00477 BC00477 V=1000.0  +MOVJ EC00477
SFTOF3D
'EndPath W3488
MOVJ C00478 BC00478 VJ=100.00  +MOVJ EC00478 VJ=100.00
'13
'Path W3489
SFTOF3D
SFTON3D P030
MOVJ C00479 BC00479 VJ=100.00  +MOVJ EC00479 VJ=100.00
SMOVL C00480 BC00480 V=800.0  +MOVJ EC00480
SMOVL C00481 BC00481 V=150.0 PL=0  +MOVJ EC00481
MACRO1 MJ#(0) ARGF9
ARCON
SWVON WEV#(10)
SFTON3D P031
SMOVL C00482 BC00482 V=12.5  +MOVJ EC00482
ARCOF
SWVOF
SMOVL C00483 BC00483 V=800.0  +MOVJ EC00483
SMOVL C00484 BC00484 V=1000.0  +MOVJ EC00484
SFTOF3D
'EndPath W3489
'Path W3490
SFTOF3D
MOVJ C00485 BC00485 VJ=100.00  +MOVJ EC00485 VJ=100.00
MACRO1 MJ#(0) ARGF6
SFTON3D P069
SMOVL C00486 BC00486 V=250.0  +MOVJ EC00486
ARCON
SMOVL C00487 BC00487 V=11.7  +MOVJ EC00487
ARCOF
SMOVL C00488 BC00488 V=250.0  +MOVJ EC00488
SFTOF3D
SFTON3D P052
MOVJ C00489 BC00489 VJ=100.00  +MOVJ EC00489 VJ=100.00
SMOVL C00490 BC00490 V=800.0  +MOVJ EC00490
SMOVL C00491 BC00491 V=150.0 PL=0  +MOVJ EC00491
MACRO1 MJ#(0) ARGF14
ARCON
SMOVL C00492 BC00492 V=10.0  +MOVJ EC00492
SMOVL C00493 BC00493 V=10.0  +MOVJ EC00493
SMOVL C00494 BC00494 V=10.0  +MOVJ EC00494
ARCOF
SMOVL C00495 BC00495 V=800.0  +MOVJ EC00495
SMOVL C00496 BC00496 V=1000.0  +MOVJ EC00496
SFTOF3D
'EndPath W3490
MOVJ C00497 BC00497 VJ=100.00  +MOVJ EC00497 VJ=100.00
'poprawic spoine - nie mialem w
'yciecia
'Path W3491
SFTOF3D
SFTON3D P053
MOVJ C00498 BC00498 VJ=100.00  +MOVJ EC00498 VJ=100.00
SMOVL C00499 BC00499 V=800.0  +MOVJ EC00499
SMOVL C00500 BC00500 V=150.0 PL=0  +MOVJ EC00500
ARCON
SMOVL C00501 BC00501 V=10.0  +MOVJ EC00501
SMOVL C00502 BC00502 V=10.0  +MOVJ EC00502
SMOVL C00503 BC00503 V=10.0  +MOVJ EC00503
ARCOF
SMOVL C00504 BC00504 V=800.0  +MOVJ EC00504
SMOVL C00505 BC00505 V=1000.0  +MOVJ EC00505
SFTOF3D
'EndPath W3491
'14
'15-brak
MOVJ C00506 BC00506 VJ=100.00  +MOVJ EC00506 VJ=100.00
'16
'Path W3491
SFTOF3D
SFTON3D P029
MOVJ C00507 BC00507 VJ=100.00  +MOVJ EC00507 VJ=100.00
SMOVL C00508 BC00508 V=800.0  +MOVJ EC00508
SMOVL C00509 BC00509 V=150.0 PL=0  +MOVJ EC00509
ARCON
SMOVL C00510 BC00510 V=10.0  +MOVJ EC00510
SMOVL C00511 BC00511 V=10.0  +MOVJ EC00511
ARCOF
SMOVL C00512 BC00512 V=800.0  +MOVJ EC00512
SMOVL C00513 BC00513 V=1000.0  +MOVJ EC00513
SFTOF3D
'EndPath W3491
MOVJ C00514 BC00514 VJ=100.00  +MOVJ EC00514 VJ=100.00
'Path W3492
SFTOF3D
SFTON3D P029
MOVJ C00515 BC00515 VJ=100.00  +MOVJ EC00515 VJ=100.00
SMOVL C00516 BC00516 V=800.0  +MOVJ EC00516
SMOVL C00517 BC00517 V=150.0 PL=0  +MOVJ EC00517
ARCON
SMOVL C00518 BC00518 V=10.0  +MOVJ EC00518
ARCOF
SMOVL C00519 BC00519 V=800.0  +MOVJ EC00519
SMOVL C00520 BC00520 V=1000.0  +MOVJ EC00520
SFTOF3D
'EndPath W3492
MOVJ C00521 BC00521 VJ=100.00  +MOVJ EC00521 VJ=100.00
MOVJ C00522 BC00522 VJ=100.00  +MOVJ EC00522 VJ=100.00
'Path W3493
SFTOF3D
SFTON3D P029
MOVJ C00523 BC00523 VJ=100.00  +MOVJ EC00523 VJ=100.00
SMOVL C00524 BC00524 V=800.0  +MOVJ EC00524
SMOVL C00525 BC00525 V=150.0 PL=0  +MOVJ EC00525
ARCON
SMOVL C00526 BC00526 V=10.0  +MOVJ EC00526
SMOVL C00527 BC00527 V=10.0  +MOVJ EC00527
SMOVL C00528 BC00528 V=10.0  +MOVJ EC00528
ARCON
SMOVL C00529 BC00529 V=11.7  +MOVJ EC00529
ARCON
SMOVL C00530 BC00530 V=11.7  +MOVJ EC00530
ARCOF
SMOVL C00531 BC00531 V=800.0  +MOVJ EC00531
SMOVL C00532 BC00532 V=1000.0  +MOVJ EC00532
SFTOF3D
'EndPath W3493
MOVJ C00533 BC00533 VJ=100.00  +MOVJ EC00533 VJ=100.00
MOVJ C00534 BC00534 VJ=100.00  +MOVJ EC00534 VJ=100.00
'17
'Path W3494
SFTOF3D
SFTON3D P027
MOVJ C00535 BC00535 VJ=100.00  +MOVJ EC00535 VJ=100.00
SMOVL C00536 BC00536 V=800.0  +MOVJ EC00536
SMOVL C00537 BC00537 V=150.0 PL=0  +MOVJ EC00537
ARCON
SMOVL C00538 BC00538 V=10.0  +MOVJ EC00538
ARCOF
SMOVL C00539 BC00539 V=800.0  +MOVJ EC00539
SMOVL C00540 BC00540 V=1000.0  +MOVJ EC00540
SFTOF3D
'EndPath W3494
'Path W3495
SFTOF3D
SFTON3D P027
MOVJ C00541 BC00541 VJ=100.00  +MOVJ EC00541 VJ=100.00
SMOVL C00542 BC00542 V=800.0  +MOVJ EC00542
SMOVL C00543 BC00543 V=150.0 PL=0  +MOVJ EC00543
ARCON
SMOVL C00544 BC00544 V=10.8  +MOVJ EC00544
ARCOF
SMOVL C00545 BC00545 V=800.0  +MOVJ EC00545
SMOVL C00546 BC00546 V=1000.0  +MOVJ EC00546
SFTOF3D
'EndPath W3495
'Path W3496
SFTOF3D
SFTON3D P027
MOVJ C00547 BC00547 VJ=100.00  +MOVJ EC00547 VJ=100.00
SFTOF3D
'EndPath W3496
MOVJ C00548 BC00548 VJ=100.00  +MOVJ EC00548 VJ=100.00
MOVJ C00549 BC00549 VJ=100.00  +MOVJ EC00549 VJ=100.00
MOVJ C00550 BC00550 VJ=100.00  +MOVJ EC00550 VJ=100.00
'18
'Path W3497
SFTOF3D
SFTON3D P024
MOVJ C00551 BC00551 VJ=100.00  +MOVJ EC00551 VJ=100.00
SMOVL C00552 BC00552 V=800.0  +MOVJ EC00552
SMOVL C00553 BC00553 V=150.0 PL=0  +MOVJ EC00553
ARCON
SMOVL C00554 BC00554 V=9.2  +MOVJ EC00554
SMOVL C00555 BC00555 V=9.2  +MOVJ EC00555
SMOVL C00556 BC00556 V=9.2  +MOVJ EC00556
SMOVL C00557 BC00557 V=9.2  +MOVJ EC00557
ARCOF
SMOVL C00558 BC00558 V=800.0  +MOVJ EC00558
SMOVL C00559 BC00559 V=1000.0  +MOVJ EC00559
SFTOF3D
'EndPath W3497
'
'Path W4855
SFTOF3D
SFTON3D P071
MOVJ C00560 BC00560 VJ=100.00  +MOVJ EC00560 VJ=100.00
SMOVL C00561 BC00561 V=800.0  +MOVJ EC00561
MACRO1 MJ#(0) ARGF9
SMOVL C00562 BC00562 V=150.0 PL=0  +MOVJ EC00562
ARCON
SMOVL C00563 BC00563 V=8.8  +MOVJ EC00563
SFTON3D P072
SMOVL C00564 BC00564 V=8.8  +MOVJ EC00564
SMOVL C00565 BC00565 V=8.8  +MOVJ EC00565
ARCOF
SMOVL C00566 BC00566 V=800.0  +MOVJ EC00566
SMOVL C00567 BC00567 V=1000.0  +MOVJ EC00567
SFTOF3D
'EndPath W4855
'
'
MOVJ C00568 BC00568 VJ=100.00  +MOVJ EC00568 VJ=100.00
'19
MOVJ C00569 BC00569 VJ=100.00  +MOVJ EC00569 VJ=100.00
'Path W3499
SFTOF3D
SFTON3D P023
MOVJ C00570 BC00570 VJ=100.00  +MOVJ EC00570 VJ=100.00
SMOVL C00571 BC00571 V=800.0  +MOVJ EC00571
SMOVL C00572 BC00572 V=150.0 PL=0  +MOVJ EC00572
MACRO1 MJ#(0) ARGF6
ARCON
SWVON WEV#(66)
SMOVL C00573 BC00573 V=7.5  +MOVJ EC00573
SMOVL C00574 BC00574 V=7.5  +MOVJ EC00574
SMOVL C00575 BC00575 V=7.5  +MOVJ EC00575
ARCOF
SWVOF
SMOVL C00576 BC00576 V=800.0  +MOVJ EC00576
SMOVL C00577 BC00577 V=1000.0  +MOVJ EC00577
SFTOF3D
'EndPath W3499
MOVJ C00578 BC00578 VJ=100.00  +MOVJ EC00578 VJ=100.00
'Path W3500
SFTOF3D
SFTON3D P034
MOVJ C00579 BC00579 VJ=100.00  +MOVJ EC00579 VJ=100.00
SMOVL C00580 BC00580 V=800.0  +MOVJ EC00580
MACRO1 MJ#(0) ARGF9
SMOVL C00581 BC00581 V=150.0 PL=0  +MOVJ EC00581
ARCON
SMOVL C00582 BC00582 V=8.3  +MOVJ EC00582
SFTON3D P050
SMOVL C00583 BC00583 V=8.3  +MOVJ EC00583
SMOVL C00584 BC00584 V=8.3  +MOVJ EC00584
ARCOF
SMOVL C00585 BC00585 V=800.0  +MOVJ EC00585
SMOVL C00586 BC00586 V=1000.0  +MOVJ EC00586
SFTOF3D
'EndPath W3500
'Path W3501
SFTOF3D
SFTON3D P051
MOVJ C00587 BC00587 VJ=100.00  +MOVJ EC00587 VJ=100.00
SMOVL C00588 BC00588 V=800.0  +MOVJ EC00588
SMOVL C00589 BC00589 V=150.0 PL=0  +MOVJ EC00589
ARCON
SWVON WEV#(60)
SMOVL C00590 BC00590 V=7.5  +MOVJ EC00590
SMOVL C00591 BC00591 V=7.5  +MOVJ EC00591
SMOVL C00592 BC00592 V=7.5  +MOVJ EC00592
ARCOF
SWVOF
SMOVL C00593 BC00593 V=800.0  +MOVJ EC00593
SMOVL C00594 BC00594 V=1000.0  +MOVJ EC00594
SFTOF3D
'EndPath W3501
MOVJ C00595 BC00595 VJ=100.00  +MOVJ EC00595 VJ=100.00
'20
MOVJ C00596 BC00596 VJ=100.00  +MOVJ EC00596 VJ=100.00
MOVJ C00597 BC00597 VJ=100.00  +MOVJ EC00597 VJ=100.00
'offset 5mm
'Path W3500
SFTOF3D
SFTON3D P032
MOVJ C00598 BC00598 VJ=100.00  +MOVJ EC00598 VJ=100.00
SMOVL C00599 BC00599 V=800.0  +MOVJ EC00599
SMOVL C00600 BC00600 V=150.0 PL=0  +MOVJ EC00600
ARCON
SMOVL C00601 BC00601 V=9.2  +MOVJ EC00601
ARCOF
SMOVL C00602 BC00602 V=800.0  +MOVJ EC00602
SMOVL C00603 BC00603 V=1000.0  +MOVJ EC00603
SFTOF3D
'EndPath W3500
SFTOF3D
'EndPath W3502
'offset 5mm
'Path W3503
SFTOF3D
SFTON3D P032
MOVJ C00604 BC00604 VJ=100.00  +MOVJ EC00604 VJ=100.00
SMOVL C00605 BC00605 V=800.0  +MOVJ EC00605
SMOVL C00606 BC00606 V=150.0 PL=0  +MOVJ EC00606
ARCON
SMOVL C00607 BC00607 V=10.0  +MOVJ EC00607
ARCOF
SMOVL C00608 BC00608 V=800.0  +MOVJ EC00608
SMOVL C00609 BC00609 V=1000.0  +MOVJ EC00609
SFTOF3D
'EndPath W3503
MOVJ C00610 BC00610 VJ=100.00  +MOVJ EC00610 VJ=100.00
'Path W3504
SFTOF3D
SFTON3D P032
MOVJ C00611 BC00611 VJ=100.00  +MOVJ EC00611 VJ=100.00
SMOVL C00612 BC00612 V=800.0  +MOVJ EC00612
SMOVL C00613 BC00613 V=150.0 PL=0  +MOVJ EC00613
ARCON
SMOVL C00614 BC00614 V=11.7  +MOVJ EC00614
SMOVL C00615 BC00615 V=11.7  +MOVJ EC00615
ARCOF
SMOVL C00616 BC00616 V=800.0  +MOVJ EC00616
SMOVL C00617 BC00617 V=1000.0  +MOVJ EC00617
SFTOF3D
'EndPath W3504
MOVJ C00618 BC00618 VJ=100.00  +MOVJ EC00618 VJ=100.00
'21
MOVJ C00619 BC00619 VJ=100.00  +MOVJ EC00619 VJ=100.00
'Path W3505
SFTOF3D
SFTON3D P021
MOVJ C00620 BC00620 VJ=100.00  +MOVJ EC00620 VJ=100.00
SMOVL C00621 BC00621 V=800.0  +MOVJ EC00621
SMOVL C00622 BC00622 V=150.0 PL=0  +MOVJ EC00622
ARCON
SFTON3D P022
SMOVL C00623 BC00623 V=10.8  +MOVJ EC00623
SMOVL C00624 BC00624 V=11.7  +MOVJ EC00624
ARCOF
SMOVL C00625 BC00625 V=800.0  +MOVJ EC00625
SMOVL C00626 BC00626 V=1000.0  +MOVJ EC00626
SFTOF3D
'EndPath W3505
MOVJ C00627 BC00627 VJ=100.00  +MOVJ EC00627 VJ=100.00
'Path W3506
SFTOF3D
SFTON3D P095
MOVJ C00628 BC00628 VJ=100.00  +MOVJ EC00628 VJ=100.00
SMOVL C00629 BC00629 V=800.0  +MOVJ EC00629
SMOVL C00630 BC00630 V=150.0 PL=0  +MOVJ EC00630
MACRO1 MJ#(0) ARGF14
ARCON
SMOVL C00631 BC00631 V=10.0  +MOVJ EC00631
SMOVL C00632 BC00632 V=10.0  +MOVJ EC00632
SMOVL C00633 BC00633 V=10.0  +MOVJ EC00633
ARCOF
SMOVL C00634 BC00634 V=800.0  +MOVJ EC00634
SMOVL C00635 BC00635 V=1000.0  +MOVJ EC00635
SFTOF3D
'EndPath W3506
'Path W3507
SFTOF3D
SFTON3D P096
MOVJ C00636 BC00636 VJ=100.00  +MOVJ EC00636 VJ=100.00
SMOVL C00637 BC00637 V=800.0  +MOVJ EC00637
SMOVL C00638 BC00638 V=150.0 PL=0  +MOVJ EC00638
SMOVL C00639 BC00639 V=10.0  +MOVJ EC00639
SMOVL C00640 BC00640 V=10.0  +MOVJ EC00640
ARCOF
SMOVL C00641 BC00641 V=800.0  +MOVJ EC00641
SMOVL C00642 BC00642 V=1000.0  +MOVJ EC00642
SFTOF3D
'EndPath W3507
MOVJ C00643 BC00643 VJ=100.00  +MOVJ EC00643 VJ=100.00
MOVJ C00644 BC00644 VJ=100.00  +MOVJ EC00644 VJ=100.00
'Path W4856
SFTOF3D
SFTON3D P071
MOVJ C00645 BC00645 VJ=100.00  +MOVJ EC00645 VJ=100.00
SMOVL C00646 BC00646 V=800.0  +MOVJ EC00646
SMOVL C00647 BC00647 V=150.0 PL=0  +MOVJ EC00647
ARCON
SMOVL C00648 BC00648 V=8.3  +MOVJ EC00648
SFTON3D P073
SMOVL C00649 BC00649 V=8.3  +MOVJ EC00649
SMOVL C00650 BC00650 V=8.3  +MOVJ EC00650
ARCOF
SMOVL C00651 BC00651 V=800.0  +MOVJ EC00651
SMOVL C00652 BC00652 V=1000.0  +MOVJ EC00652
SFTOF3D
'EndPath W4856
MOVJ C00653 BC00653 VJ=100.00  +MOVJ EC00653 VJ=100.00
MOVJ C00654 BC00654 VJ=100.00  +MOVJ EC00654 VJ=100.00
'cut_wire_dol
'cut_wire_dol
'cut_wire_dol
CALL JOB:CLEAN-R1_KM_NEW
MOVJ C00655 BC00655 VJ=100.00  +MOVJ EC00655 VJ=100.00
MOVJ C00656 BC00656 VJ=100.00  +MOVJ EC00656 VJ=100.00
MOVJ C00657 BC00657 VJ=100.00  +MOVJ EC00657 VJ=100.00
'Path S4011
SFTOF3D
MOVJ C00658 BC00658 VJ=100.00  +MOVJ EC00658 VJ=100.00
MOVL C00659 BC00659 V=666.7  +MOVJ EC00659 VJ=100.00
SMOVL C00660 BC00660 V=166.7  +MOVJ EC00660
SREFP 3 C00661 BC00661  +REFP EC00661
CALL JOB:SEARCH-R1-S13D
SET P049 P006
SFTON3D P049
SMOVL C00662 BC00662 V=166.7  +MOVJ EC00662
SMOVL C00663 BC00663 V=166.7  +MOVJ EC00663
SREFP 3 C00664 BC00664  +REFP EC00664
CALL JOB:SEARCH-R1-S13D
SET P049 P006
SFTON3D P049
SMOVL C00665 BC00665 V=166.7  +MOVJ EC00665
SMOVL C00666 BC00666 V=166.7  +MOVJ EC00666
SMOVL C00667 BC00667 V=166.7  +MOVJ EC00667
SREFP 3 C00668 BC00668  +REFP EC00668
CALL JOB:SEARCH-R1-S13D
SET P049 P006
SFTON3D P049
SMOVL C00669 BC00669 V=166.7  +MOVJ EC00669
MOVL C00670 BC00670 V=1000.0  +MOVJ EC00670 VJ=100.00
'EndPath S4011
'Path S4010
SFTOF3D
MOVJ C00671 BC00671 VJ=100.00  +MOVJ EC00671 VJ=100.00
SMOVL C00672 BC00672 V=666.7  +MOVJ EC00672
SMOVL C00673 BC00673 V=166.7  +MOVJ EC00673
SREFP 3 C00674 BC00674  +REFP EC00674
CALL JOB:SEARCH-R1-S13D
SET P048 P006
SFTON3D P048
SMOVL C00675 BC00675 V=166.7  +MOVJ EC00675
SMOVL C00676 BC00676 V=166.7  +MOVJ EC00676
SREFP 3 C00677 BC00677  +REFP EC00677
CALL JOB:SEARCH-R1-S13D
SET P048 P006
SFTON3D P048
SMOVL C00678 BC00678 V=233.3  +MOVJ EC00678
MOVL C00679 BC00679 V=1000.0  +MOVJ EC00679 VJ=100.00
'EndPath S4010
'Path S4009
SFTOF3D
MOVJ C00680 BC00680 VJ=100.00  +MOVJ EC00680 VJ=100.00
MOVL C00681 BC00681 V=666.7  +MOVJ EC00681 VJ=100.00
SMOVL C00682 BC00682 V=166.7  +MOVJ EC00682
SREFP 3 C00683 BC00683  +REFP EC00683
CALL JOB:SEARCH-R1-S13D
SET P047 P006
SFTON3D P047
SMOVL C00684 BC00684 V=166.7  +MOVJ EC00684
SMOVL C00685 BC00685 V=166.7  +MOVJ EC00685
SREFP 3 C00686 BC00686  +REFP EC00686
CALL JOB:SEARCH-R1-S13D
SET P047 P006
SFTON3D P047
SMOVL C00687 BC00687 V=166.7  +MOVJ EC00687
MOVL C00688 BC00688 V=1000.0  +MOVJ EC00688 VJ=100.00
'EndPath S4009
MOVJ C00689 BC00689 VJ=100.00  +MOVJ EC00689 VJ=100.00
'Path S4008
SFTOF3D
MOVJ C00690 BC00690 VJ=100.00  +MOVJ EC00690 VJ=100.00
MOVL C00691 BC00691 V=1000.0  +MOVJ EC00691 VJ=100.00
'EndPath S4008
'Path S4007
SFTOF3D
MOVJ C00692 BC00692 VJ=100.00  +MOVJ EC00692 VJ=100.00
MOVL C00693 BC00693 V=666.7  +MOVJ EC00693 VJ=100.00
SMOVL C00694 BC00694 V=166.7  +MOVJ EC00694
SREFP 3 C00695 BC00695  +REFP EC00695
CALL JOB:SEARCH-R1-S13D
SET P045 P006
SFTON3D P045
SMOVL C00696 BC00696 V=166.7  +MOVJ EC00696
SMOVL C00697 BC00697 V=166.7  +MOVJ EC00697
SMOVL C00698 BC00698 V=166.7  +MOVJ EC00698
SREFP 3 C00699 BC00699  +REFP EC00699
CALL JOB:SEARCH-R1-S13D
SET P045 P006
SFTON3D P045
SMOVL C00700 BC00700 V=166.7  +MOVJ EC00700
MOVL C00701 BC00701 V=1000.0  +MOVJ EC00701 VJ=100.00
'EndPath S4007
'Path S3506
SFTOF3D
MOVJ C00702 BC00702 VJ=100.00  +MOVJ EC00702 VJ=100.00
MOVL C00703 BC00703 V=666.7  +MOVJ EC00703 VJ=100.00
SMOVL C00704 BC00704 V=166.7  +MOVJ EC00704
SREFP 3 C00705 BC00705  +REFP EC00705
CALL JOB:SEARCH-R1-S13D
SET P044 P006
SFTON3D P044
SMOVL C00706 BC00706 V=166.7  +MOVJ EC00706
SMOVL C00707 BC00707 V=166.7  +MOVJ EC00707
SREFP 3 C00708 BC00708  +REFP EC00708
CALL JOB:SEARCH-R1-S13D
SET P044 P006
SFTON3D P044
SFTOF3D
SMOVL C00709 BC00709 V=166.7  +MOVJ EC00709
MOVL C00710 BC00710 V=1000.0  +MOVJ EC00710 VJ=100.00
'EndPath S3506
MOVJ C00711 BC00711 VJ=100.00  +MOVJ EC00711 VJ=100.00
MOVJ C00712 BC00712 VJ=50.00  +MOVJ EC00712 VJ=50.00
MOVJ C00713 BC00713 VJ=50.00  +MOVJ EC00713 VJ=50.00
MOVJ C00714 BC00714 VJ=100.00  +MOVJ EC00714 VJ=100.00
MOVJ C00715 BC00715 VJ=100.00  +MOVJ EC00715 VJ=100.00
MOVJ C00716 BC00716 VJ=100.00  +MOVJ EC00716 VJ=100.00
MOVJ C00717 BC00717 VJ=100.00  +MOVJ EC00717 VJ=100.00
'Path S4006
SFTOF3D
MOVJ C00718 BC00718 VJ=100.00  +MOVJ EC00718 VJ=100.00
MOVL C00719 BC00719 V=666.7  +MOVJ EC00719 VJ=100.00
SMOVL C00720 BC00720 V=166.7  +MOVJ EC00720
SREFP 3 C00721 BC00721  +REFP EC00721
CALL JOB:SEARCH-R1-S13D
SET P043 P006
SFTON3D P043
SMOVL C00722 BC00722 V=166.7  +MOVJ EC00722
SMOVL C00723 BC00723 V=166.7  +MOVJ EC00723
SMOVL C00724 BC00724 V=166.7  +MOVJ EC00724
SREFP 3 C00725 BC00725  +REFP EC00725
CALL JOB:SEARCH-R1-S13D
SET P043 P006
SFTON3D P043
SMOVL C00726 BC00726 V=166.7  +MOVJ EC00726
MOVL C00727 BC00727 V=1000.0  +MOVJ EC00727 VJ=100.00
'EndPath S4006
'Path S4005
SFTOF3D
MOVJ C00728 BC00728 VJ=100.00  +MOVJ EC00728 VJ=100.00
MOVL C00729 BC00729 V=800.0  +MOVJ EC00729 VJ=100.00
SMOVL C00730 BC00730 V=166.7  +MOVJ EC00730
SREFP 3 C00731 BC00731  +REFP EC00731
CALL JOB:SEARCH-R1-S13D
SET P042 P006
SFTON3D P042
SMOVL C00732 BC00732 V=166.7  +MOVJ EC00732
SMOVL C00733 BC00733 V=166.7  +MOVJ EC00733
SREFP 3 C00734 BC00734  +REFP EC00734
CALL JOB:SEARCH-R1-S13D
SET P042 P006
SFTON3D P042
SMOVL C00735 BC00735 V=166.7  +MOVJ EC00735
MOVL C00736 BC00736 V=1000.0  +MOVJ EC00736 VJ=100.00
'EndPath S4005
'Path S4004
SFTOF3D
MOVJ C00737 BC00737 VJ=100.00  +MOVJ EC00737 VJ=100.00
MOVL C00738 BC00738 V=800.0  +MOVJ EC00738 VJ=100.00
SMOVL C00739 BC00739 V=166.7  +MOVJ EC00739
SMOVL C00740 BC00740 V=166.7  +MOVJ EC00740
SREFP 3 C00741 BC00741  +REFP EC00741
CALL JOB:SEARCH-R1-S13D
SET P041 P006
SFTON3D P041
SMOVL C00742 BC00742 V=166.7  +MOVJ EC00742
SMOVL C00743 BC00743 V=166.7  +MOVJ EC00743
SREFP 3 C00744 BC00744  +REFP EC00744
CALL JOB:SEARCH-R1-S13D
SET P041 P006
SFTON3D P041
SMOVL C00745 BC00745 V=166.7  +MOVJ EC00745
SREFP 3 C00746 BC00746  +REFP EC00746
CALL JOB:SEARCH-R1-S13D
SET P041 P006
SFTON3D P041
SMOVL C00747 BC00747 V=166.7  +MOVJ EC00747
MOVL C00748 BC00748 V=1000.0  +MOVJ EC00748 VJ=100.00
'EndPath S4004
'Path S4003
SFTOF3D
MOVJ C00749 BC00749 VJ=100.00  +MOVJ EC00749 VJ=100.00
MOVL C00750 BC00750 V=800.0  +MOVJ EC00750 VJ=100.00
SMOVL C00751 BC00751 V=166.7  +MOVJ EC00751
SREFP 3 C00752 BC00752  +REFP EC00752
CALL JOB:SEARCH-R1-S13D
SET P040 P006
SFTON3D P040
SMOVL C00753 BC00753 V=250.0  +MOVJ EC00753
SMOVL C00754 BC00754 V=250.0  +MOVJ EC00754
SMOVL C00755 BC00755 V=166.7  +MOVJ EC00755
SREFP 3 C00756 BC00756  +REFP EC00756
CALL JOB:SEARCH-R1-S13D
SET P040 P006
SFTON3D P040
SMOVL C00757 BC00757 V=166.7  +MOVJ EC00757
SMOVL C00758 BC00758 V=166.7  +MOVJ EC00758
SREFP 3 C00759 BC00759  +REFP EC00759
CALL JOB:SEARCH-R1-S13D
SET P040 P006
SFTON3D P040
SMOVL C00760 BC00760 V=166.7  +MOVJ EC00760
MOVL C00761 BC00761 V=1000.0  +MOVJ EC00761 VJ=100.00
'EndPath S4003
'Path W4012
SFTOF3D
SFTON3D P040
MOVJ C00762 BC00762 VJ=100.00  +MOVJ EC00762 VJ=100.00
SMOVL C00763 BC00763 V=800.0  +MOVJ EC00763
SMOVL C00764 BC00764 V=150.0 PL=0  +MOVJ EC00764
ARCON
SMOVL C00765 BC00765 V=11.7  +MOVJ EC00765
ARCOF
SMOVL C00766 BC00766 V=800.0  +MOVJ EC00766
SMOVL C00767 BC00767 V=1000.0  +MOVJ EC00767
SFTOF3D
'EndPath W4012
'Path W4013
SFTOF3D
SFTON3D P040
MOVJ C00768 BC00768 VJ=100.00  +MOVJ EC00768 VJ=100.00
SMOVL C00769 BC00769 V=800.0  +MOVJ EC00769
SMOVL C00770 BC00770 V=150.0 PL=0  +MOVJ EC00770
ARCON
SMOVL C00771 BC00771 V=10.0  +MOVJ EC00771
ARCOF
SMOVL C00772 BC00772 V=800.0  +MOVJ EC00772
SMOVL C00773 BC00773 V=1000.0  +MOVJ EC00773
SMOVL C00774 BC00774 V=1000.0  +MOVJ EC00774
SFTOF3D
'EndPath W4013
'Path W4014
SFTOF3D
SFTON3D P040
MOVJ C00775 BC00775 VJ=100.00  +MOVJ EC00775 VJ=100.00
SMOVL C00776 BC00776 V=800.0  +MOVJ EC00776
SMOVL C00777 BC00777 V=150.0 PL=0  +MOVJ EC00777
ARCON
SMOVL C00778 BC00778 V=10.0  +MOVJ EC00778
ARCOF
SMOVL C00779 BC00779 V=800.0  +MOVJ EC00779
SMOVL C00780 BC00780 V=1000.0  +MOVJ EC00780
SFTOF3D
'EndPath W4014
'
MOVJ C00781 BC00781 VJ=100.00  +MOVJ EC00781 VJ=100.00
MOVJ C00782 BC00782 VJ=100.00  +MOVJ EC00782 VJ=100.00
MOVJ C00783 BC00783 VJ=100.00  +MOVJ EC00783 VJ=100.00
MOVJ C00784 BC00784 VJ=100.00  +MOVJ EC00784 VJ=100.00
MOVJ C00785 BC00785 VJ=100.00  +MOVJ EC00785 VJ=100.00
'Path W3522
SFTOF3D
SFTON3D P045
MOVJ C00786 BC00786 VJ=100.00  +MOVJ EC00786 VJ=100.00
SMOVL C00787 BC00787 V=800.0  +MOVJ EC00787
SMOVL C00788 BC00788 V=150.0 PL=0  +MOVJ EC00788
MACRO1 MJ#(0) ARGF9
ARCON
SMOVL C00789 BC00789 V=11.7  +MOVJ EC00789
ARCOF
SMOVL C00790 BC00790 V=800.0  +MOVJ EC00790
SMOVL C00791 BC00791 V=1000.0  +MOVJ EC00791
SFTOF3D
'EndPath W3522
'Path W3520
SFTOF3D
SFTON3D P044
MOVJ C00792 BC00792 VJ=100.00  +MOVJ EC00792 VJ=100.00
SMOVL C00793 BC00793 V=800.0  +MOVJ EC00793
SMOVL C00794 BC00794 V=166.7 PL=0  +MOVJ EC00794
ARCON
SMOVL C00795 BC00795 V=11.7  +MOVJ EC00795
SMOVL C00796 BC00796 V=11.7  +MOVJ EC00796
SMOVL C00797 BC00797 V=11.7  +MOVJ EC00797
ARCOF
SMOVL C00798 BC00798 V=800.0  +MOVJ EC00798
SMOVL C00799 BC00799 V=1000.0  +MOVJ EC00799
SFTOF3D
SFTOF3D
'EndPath W3519
'1
MOVJ C00800 BC00800 VJ=100.00  +MOVJ EC00800 VJ=100.00
MOVJ C00801 BC00801 VJ=100.00  +MOVJ EC00801 VJ=100.00
'Path W3509
SFTOF3D
SFTON3D P048
MOVJ C00802 BC00802 VJ=100.00  +MOVJ EC00802 VJ=100.00
SMOVL C00803 BC00803 V=800.0  +MOVJ EC00803
SMOVL C00804 BC00804 V=150.0 PL=0  +MOVJ EC00804
ARCON
SMOVL C00805 BC00805 V=11.7  +MOVJ EC00805
ARCOF
SMOVL C00806 BC00806 V=800.0  +MOVJ EC00806
SFTOF3D
'EndPath W3509
'Path W3510
SFTOF3D
SFTON3D P049
MOVJ C00807 BC00807 VJ=100.00  +MOVJ EC00807 VJ=100.00
SMOVL C00808 BC00808 V=800.0  +MOVJ EC00808
SMOVL C00809 BC00809 V=150.0 PL=0  +MOVJ EC00809
MACRO1 MJ#(0) ARGF6
ARCON
SMOVL C00810 BC00810 V=9.2  +MOVJ EC00810
SMOVL C00811 BC00811 V=9.2  +MOVJ EC00811
SMOVL C00812 BC00812 V=9.2  +MOVJ EC00812
SMOVL C00813 BC00813 V=9.2  +MOVJ EC00813
SMOVL C00814 BC00814 V=9.2  +MOVJ EC00814
ARCOF
MOVJ C00815 BC00815 VJ=30.00  +MOVJ EC00815 VJ=80.00
MOVJ C00816 BC00816 VJ=30.00  +MOVJ EC00816 VJ=30.00
SMOVL C00817 BC00817 V=166.7  +MOVJ EC00817
ARCON
SMOVL C00818 BC00818 V=13.3  +MOVJ EC00818
SMOVL C00819 BC00819 V=13.3  +MOVJ EC00819
SMOVL C00820 BC00820 V=13.3  +MOVJ EC00820
ARCOF
SMOVL C00821 BC00821 V=333.3  +MOVJ EC00821
SMOVL C00822 BC00822 V=666.7  +MOVJ EC00822
SMOVL C00823 BC00823 V=166.7  +MOVJ EC00823
ARCON
SMOVL C00824 BC00824 V=13.3  +MOVJ EC00824
SMOVL C00825 BC00825 V=12.5  +MOVJ EC00825
SMOVL C00826 BC00826 V=12.5  +MOVJ EC00826
ARCOF
SFTOF3D
SMOVL C00827 BC00827 V=250.0  +MOVJ EC00827
'EndPath W3510
MOVJ C00828 BC00828 VJ=100.00  +MOVJ EC00828 VJ=100.00
'2
MOVJ C00829 BC00829 VJ=100.00  +MOVJ EC00829 VJ=100.00
MOVJ C00830 BC00830 VJ=100.00  +MOVJ EC00830 VJ=100.00
MOVJ C00831 BC00831 VJ=100.00  +MOVJ EC00831 VJ=100.00
'Path W3511
SFTOF3D
SFTON3D P043
MOVJ C00832 BC00832 VJ=100.00  +MOVJ EC00832 VJ=100.00
SMOVL C00833 BC00833 V=800.0  +MOVJ EC00833
SMOVL C00834 BC00834 V=166.7 PL=0  +MOVJ EC00834
MACRO1 MJ#(0) ARGF9
ARCON
SMOVL C00835 BC00835 V=11.7  +MOVJ EC00835
ARCOF
SMOVL C00836 BC00836 V=800.0  +MOVJ EC00836
SMOVL C00837 BC00837 V=1000.0  +MOVJ EC00837
SFTOF3D
'EndPath W3511
'Path W3512
SFTOF3D
SFTON3D P042
MOVJ C00838 BC00838 VJ=100.00  +MOVJ EC00838 VJ=100.00
SMOVL C00839 BC00839 V=800.0  +MOVJ EC00839
SMOVL C00840 BC00840 V=150.0 PL=0  +MOVJ EC00840
ARCON
SMOVL C00841 BC00841 V=11.7  +MOVJ EC00841
ARCOF
SMOVL C00842 BC00842 V=800.0  +MOVJ EC00842
SMOVL C00843 BC00843 V=1000.0  +MOVJ EC00843
SFTOF3D
'EndPath W3512
'3
MOVJ C00844 BC00844 VJ=100.00  +MOVJ EC00844 VJ=100.00
MOVJ C00845 BC00845 VJ=100.00  +MOVJ EC00845 VJ=100.00
MOVJ C00846 BC00846 VJ=100.00  +MOVJ EC00846 VJ=100.00
MOVJ C00847 BC00847 VJ=100.00  +MOVJ EC00847 VJ=100.00
'Path W3514
SFTOF3D
SFTON3D P047
MOVJ C00848 BC00848 VJ=100.00  +MOVJ EC00848 VJ=100.00
SMOVL C00849 BC00849 V=800.0  +MOVJ EC00849
SMOVL C00850 BC00850 V=150.0 PL=0  +MOVJ EC00850
ARCON
SMOVL C00851 BC00851 V=11.7  +MOVJ EC00851
ARCOF
SMOVL C00852 BC00852 V=800.0  +MOVJ EC00852
SMOVL C00853 BC00853 V=1000.0  +MOVJ EC00853
SFTOF3D
'EndPath W3514
'Path W3518
SFTOF3D
SFTON3D P047
MOVJ C00854 BC00854 VJ=100.00  +MOVJ EC00854 VJ=100.00
SMOVL C00855 BC00855 V=800.0  +MOVJ EC00855
SMOVL C00856 BC00856 V=150.0 PL=0  +MOVJ EC00856
ARCON
SMOVL C00857 BC00857 V=11.7  +MOVJ EC00857
ARCOF
SMOVL C00858 BC00858 V=800.0  +MOVJ EC00858
SMOVL C00859 BC00859 V=1000.0  +MOVJ EC00859
SFTOF3D
'EndPath W3518
MOVJ C00860 BC00860 VJ=100.00  +MOVJ EC00860 VJ=100.00
MOVJ C00861 BC00861 VJ=100.00  +MOVJ EC00861 VJ=100.00
MOVJ C00862 BC00862 VJ=100.00  +MOVJ EC00862 VJ=100.00
MOVJ C00863 BC00863 VJ=100.00  +MOVJ EC00863 VJ=100.00
'Path W3516
SFTOF3D
SFTON3D P043
MOVJ C00864 BC00864 VJ=50.00  +MOVJ EC00864 VJ=50.00
MOVJ C00865 BC00865 VJ=100.00  +MOVJ EC00865 VJ=100.00
SMOVL C00866 BC00866 V=800.0  +MOVJ EC00866
SMOVL C00867 BC00867 V=150.0 PL=0  +MOVJ EC00867
ARCON
SMOVL C00868 BC00868 V=11.7  +MOVJ EC00868
ARCOF
SMOVL C00869 BC00869 V=800.0  +MOVJ EC00869
SMOVL C00870 BC00870 V=1000.0  +MOVJ EC00870
SFTOF3D
'EndPath W3516
'Path W3515
SFTOF3D
SFTON3D P042
MOVJ C00871 BC00871 VJ=100.00  +MOVJ EC00871 VJ=100.00
SMOVL C00872 BC00872 V=800.0  +MOVJ EC00872
SMOVL C00873 BC00873 V=166.7 PL=0  +MOVJ EC00873
ARCON
SMOVL C00874 BC00874 V=10.8  +MOVJ EC00874
ARCOF
SMOVL C00875 BC00875 V=800.0  +MOVJ EC00875
SMOVL C00876 BC00876 V=1000.0  +MOVJ EC00876
SFTOF3D
'EndPath W3515
MOVJ C00877 BC00877 VJ=100.00  +MOVJ EC00877 VJ=100.00
MOVJ C00878 BC00878 VJ=100.00  +MOVJ EC00878 VJ=100.00
MOVJ C00879 BC00879 VJ=100.00  +MOVJ EC00879 VJ=100.00
MOVJ C00880 BC00880 VJ=100.00  +MOVJ EC00880 VJ=100.00
'Path W3523
SFTOF3D
SFTON3D P046
MOVJ C00881 BC00881 VJ=100.00  +MOVJ EC00881 VJ=100.00
SMOVL C00882 BC00882 V=800.0  +MOVJ EC00882
SMOVL C00883 BC00883 V=166.7 PL=0  +MOVJ EC00883
MACRO1 MJ#(0) ARGF14
ARCON
SMOVL C00884 BC00884 V=10.0  +MOVJ EC00884
ARCOF
SMOVL C00885 BC00885 V=800.0  +MOVJ EC00885
SMOVL C00886 BC00886 V=1000.0  +MOVJ EC00886
SFTOF3D
'EndPath W3523
'Path W4015
SFTOF3D
SFTON3D P044
MOVJ C00887 BC00887 VJ=100.00  +MOVJ EC00887 VJ=100.00
SMOVL C00888 BC00888 V=800.0  +MOVJ EC00888
SMOVL C00889 BC00889 V=150.0 PL=0  +MOVJ EC00889
MACRO1 MJ#(0) ARGF9
ARCON
SMOVL C00890 BC00890 V=10.8  +MOVJ EC00890
ARCOF
SMOVL C00891 BC00891 V=800.0  +MOVJ EC00891
SMOVL C00892 BC00892 V=1000.0  +MOVJ EC00892
SFTOF3D
'EndPath W4015
MOVJ C00893 BC00893 VJ=100.00  +MOVJ EC00893 VJ=100.00
MOVJ C00894 BC00894 VJ=100.00  +MOVJ EC00894 VJ=100.00
MOVJ C00895 BC00895 VJ=100.00  +MOVJ EC00895 VJ=100.00
MOVJ C00896 BC00896 VJ=100.00  +MOVJ EC00896 VJ=100.00
'Path W4016
SFTOF3D
SFTON3D P041
MOVJ C00897 BC00897 VJ=100.00  +MOVJ EC00897 VJ=100.00
SMOVL C00898 BC00898 V=800.0  +MOVJ EC00898
SMOVL C00899 BC00899 V=150.0 PL=0  +MOVJ EC00899
MACRO1 MJ#(0) ARGF14
ARCON
SMOVL C00900 BC00900 V=10.0  +MOVJ EC00900
SMOVL C00901 BC00901 V=10.0  +MOVJ EC00901
SMOVL C00902 BC00902 V=10.0  +MOVJ EC00902
ARCOF
SMOVL C00903 BC00903 V=800.0  +MOVJ EC00903
SMOVL C00904 BC00904 V=1000.0  +MOVJ EC00904
SFTOF3D
MOVJ C00905 BC00905 VJ=100.00  +MOVJ EC00905 VJ=100.00
MOVJ C00906 BC00906 VJ=100.00  +MOVJ EC00906 VJ=100.00
MOVJ C00907 BC00907 VJ=100.00  +MOVJ EC00907 VJ=100.00
MOVJ C00908 BC00908 VJ=100.00  +MOVJ EC00908 VJ=100.00
MOVJ C00909 BC00909 VJ=100.00  +MOVJ EC00909 VJ=100.00
END
